// Basic passive two-threshold pneumatic-pressure CM. Both switches active is
// implausible and faults with both exact tags; neither/high-only are status states.
FUNCTION_BLOCK FB_AirPressureMonitorCM EXTENDS FB_ControlModuleBase
VAR_INPUT
    ParCfg : ST_AirPressureParCfg;
    ParCmd : ST_AirPressureParCmd;
END_VAR
VAR_OUTPUT
    OutCmd : ST_AirPressureOutCmd;
    OutImm : ST_AirPressureOutImm;
END_VAR
VAR
    {attribute 'OPC.UA.DA' := '0'}
    _hal : REFERENCE TO ST_AirPressureHal;
    _lowIdentity, _operatingIdentity : ST_IoPointIdentity;
    _bothTags, _bothAddresses : STRING(80);
    // Both switches reading active is only a genuine wiring/sensor fault when it
    // PERSISTS. The two mechanical switches trip at different pressures and have
    // their own response delays, so while the system pressurises a brief overlap
    // is normal physics, not a defect. Because the fault latches (an operator
    // reset is required to clear it), a single spurious cycle would otherwise
    // block Control On indefinitely — observed on the press, where the sensors
    // read consistently in steady state yet the conflict fault stayed raised.
    // Same idiom as ST_ConfigurableCylinderParCfg.DiscrepancyTime.
    _conflictTimer : TON;
END_VAR
VAR PERSISTENT
    // §3.8a/§3.8b — deployment data: editable from the HMI, retained across
    // a restart, and never part of a model recipe. The Setup registration,
    // not this declaration, is what permits a write (§3.10.2).
    StationCfg : ST_AirPressureStationCfg;
END_VAR

Cyclic();

METHOD Setup : BOOL
VAR_INPUT
    Name : STRING(80);
    HalRef : REFERENCE TO ST_AirPressureHal;
END_VAR
_M_SetName(Name);
_M_SetPresentation(DisplayNameKey := 'std.moduleType.airPressure.name',
    DescriptionKey := 'std.moduleType.airPressure.description',
    TypeKey := 'std.moduleType.airPressure');
_hal REF= HalRef;
// §3.8b — a retained image from an unrecognized layout is re-initialized,
// never interpreted by field position. Version 0 is a first boot: nothing
// was retained, so nothing was lost and nothing is announced.
IF StationCfg.SchemaVersion <> 1 THEN
    StationCfg.SchemaVersion := 1;
    StationCfg.ConflictTime := T#500MS;
END_IF
// §3.10.2 — publish the one value a commissioning engineer tunes here.
// READY is required: re-timing fault qualification underneath a running
// cycle would change what counts as a fault while it is being judged.
Setup := __ISVALIDREF(_hal)
    AND M_RegisterConfigDuration(Key := 'airPressure.conflictTime',
        Item := 'StationCfg/ConflictTime',
        LabelKey := 'std.config.airPressure.conflictTime',
        Kind := E_ConfigKind.STATION_CFG,
        pTarget := ADR(StationCfg.ConflictTime),
        MinimumMs := 0, MaximumMs := 10000,
        RequiresReady := TRUE);
END_METHOD

METHOD ConfigureIoIdentity
VAR_INPUT
    LowSensor : ST_IoPointIdentity;
    OperatingSensor : ST_IoPointIdentity;
END_VAR
_lowIdentity := LowSensor;
_operatingIdentity := OperatingSensor;
_bothTags := CONCAT(LowSensor.Tag, CONCAT(' / ', OperatingSensor.Tag));
_bothAddresses := CONCAT(LowSensor.Address, CONCAT(' / ', OperatingSensor.Address));
END_METHOD

METHOD PROTECTED OnCyclic : DINT
OnCyclic := SUPER^.OnCyclic();
IF __ISVALIDREF(_hal) THEN
    OutImm.LowPressure := _hal.LowPressure;
    OutImm.OperatingPressure := _hal.OperatingPressure;
    OutImm.Quality := _hal.Quality;
    // Qualify the conflict over StationCfg.ConflictTime before treating it as
    // a fault, so the transient overlap seen while air fills cannot latch a
    // permanent fault.
    _conflictTimer(IN := _hal.LowPressure AND _hal.OperatingPressure,
        PT := StationCfg.ConflictTime);
    OutImm.Contradictory := _conflictTimer.Q;
    OutImm.PressureOk := _hal.OperatingPressure AND NOT _hal.LowPressure AND _hal.Quality;
    IF OutImm.Contradictory THEN
        _M_FaultIoN(Code := PL_ModuleReasons.AIR_SWITCH_CONFLICT,
            Text := 'std.error.airPressureSwitchConflict',
            IoTag := _bothTags, IoAddress := _bothAddresses);
    END_IF
ELSE
    OutImm.LowPressure := FALSE;
    OutImm.OperatingPressure := FALSE;
    OutImm.Quality := FALSE;
    OutImm.Contradictory := FALSE;
    OutImm.PressureOk := FALSE;
END_IF
OutImm.LowSensorTag := _lowIdentity.Tag;
OutImm.OperatingSensorTag := _operatingIdentity.Tag;
OutImm.Diagnostic := Status.Diagnostic;
END_METHOD

METHOD PROTECTED _M_Dispatch
_M_Fault(E_Reason.UNSUPPORTED_COMMAND,
    'std.error.passiveInputHasNoCommand');
END_METHOD

METHOD PROTECTED _M_PublishStatus
SUPER^._M_PublishStatus();
OutImm.Diagnostic := Status.Diagnostic;
END_METHOD

END_FUNCTION_BLOCK

(* stored: Version 1.1.0.1, ProductVersion 3.1.4024.12
   POU FB_AirPressureMonitorCM: Id {1862918e-aa03-4414-ac9d-d7a19314762e}, SpecialFunc None
   Method Setup: Id {9affcfde-9e41-401a-bfe2-d67dc9795c5c}
   Method ConfigureIoIdentity: Id {825e28ad-8325-464e-9a73-2d407b04b0fc}
   Method OnCyclic: Id {9a04f407-a329-426e-992c-0f0f27ee5b78}
   Method _M_Dispatch: Id {c1ed801c-d79c-4e7d-be30-b7129ae3fb84}
   Method _M_PublishStatus: Id {fc69255d-7bf9-4132-964d-3ecb5983d52f} *)
